PROGRAM ObserverPatternTest
VAR
	machine: VisitorHandler;
	AlarmLogger1: AlarmLogger;
	AlarmLogger2: AlarmLogger;
	AttachAlarmLogger1: BOOL;
	AttachAlarmLogger2: BOOL;
	DetachAlarmLogger1: BOOL;
	DetachAlarmLogger2: BOOL;
END_VAR

IF AttachAlarmLogger1 THEN
	AttachAlarmLogger1:= FALSE;
	machine.subscribe(AlarmLogger1);
END_IF


IF AttachAlarmLogger2 THEN
	AttachAlarmLogger2:= FALSE;
	machine.subscribe(AlarmLogger2);
END_IF


IF DetachAlarmLogger1 THEN
	DetachAlarmLogger1:= FALSE;
	machine.unSubscribe(AlarmLogger1);
END_IF

IF DetachAlarmLogger2 THEN
	DetachAlarmLogger2:= FALSE;
	machine.unSubscribe(AlarmLogger2);
END_IF



Machine.notify();
Machine.simulateValue();

END_PROGRAM

(* stored: Version 1.1.0.1
   POU ObserverPatternTest: Id {534f6ce9-3e97-41da-ab91-116f7415a188}, SpecialFunc None *)
